// TwinCAT 3 PLC project IORead
// ProgramVersion: 3.1.4024.12
// libraries:
//   Tc2_Standard, * (Beckhoff Automation GmbH)
//   Tc2_System, * (Beckhoff Automation GmbH)
//   Tc3_Module, * (Beckhoff Automation GmbH)
// project tree:
//   DUTs/ StReadIO.TcDUT
//   GVLs/ IO.TcGVL
//   / PlcTask.TcTTO
//   POUs/ MAIN.TcPOU, SystemTest.TcPOU
// real-time tasks:
//   TASK PlcTask: cycle T#10ms, priority 20, ADS port 350

CONFIGURATION IORead
    RESOURCE PLC ON TwinCAT3
        TASK PlcTask(INTERVAL := T#10ms, PRIORITY := 20);
        PROGRAM MAIN WITH PlcTask : MAIN;
    END_RESOURCE
END_CONFIGURATION

// ---- DUTs/StReadIO.TcDUT
TYPE StReadIO :
STRUCT
	{attribute addProperty Name "<#Actual IO Staus #>"}
	st_ReadIO : BOOL;
END_STRUCT
END_TYPE

// ---- GVLs/IO.TcGVL
{attribute 'qualified_only'}
VAR_GLOBAL
	g_ReadIO AT %I* : BOOL;
END_VAR

// ---- POUs/MAIN.TcPOU
PROGRAM MAIN
VAR
	MainReadIO : StReadIO;
	FB_SystemTest : SystemTest;
END_VAR

FB_SystemTest();

MainReadIO.st_ReadIO := IO.g_ReadIO;

END_PROGRAM

// ---- POUs/SystemTest.TcPOU
FUNCTION_BLOCK SystemTest
VAR_INPUT
END_VAR
VAR_OUTPUT
END_VAR
VAR
END_VAR

IF IO.g_ReadIO THEN
	IO.g_ReadIO := FALSE;
ELSE
	IO.g_ReadIO := TRUE;
END_IF

END_FUNCTION_BLOCK
